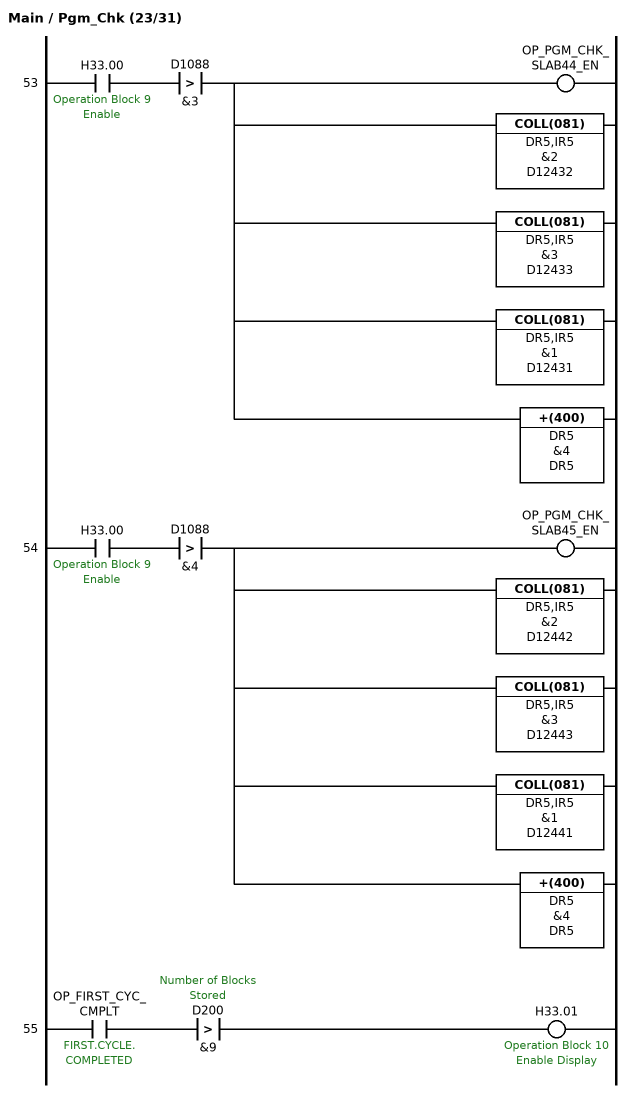
; [picture p120: Main / Pgm_Chk, rungs 53-55]
; rung 53
LD H33.00  ; Operation Block 9 Enable
AND>(320) D1088 &3
OUT OP_PGM_CHK_SLAB44_EN
COLL(081) DR5,IR5 &2 D12432
COLL(081) DR5,IR5 &3 D12433
COLL(081) DR5,IR5 &1 D12431
+(400) DR5 &4 DR5
; rung 54
LD H33.00  ; Operation Block 9 Enable
AND>(320) D1088 &4
OUT OP_PGM_CHK_SLAB45_EN
COLL(081) DR5,IR5 &2 D12442
COLL(081) DR5,IR5 &3 D12443
COLL(081) DR5,IR5 &1 D12441
+(400) DR5 &4 DR5
; rung 55
LD OP_FIRST_CYC_CMPLT  ; FIRST.CYCLE.COMPLETED
AND>(320) D200 &9  ; Number of Blocks Stored
OUT H33.01  ; Operation Block 10 Enable Display

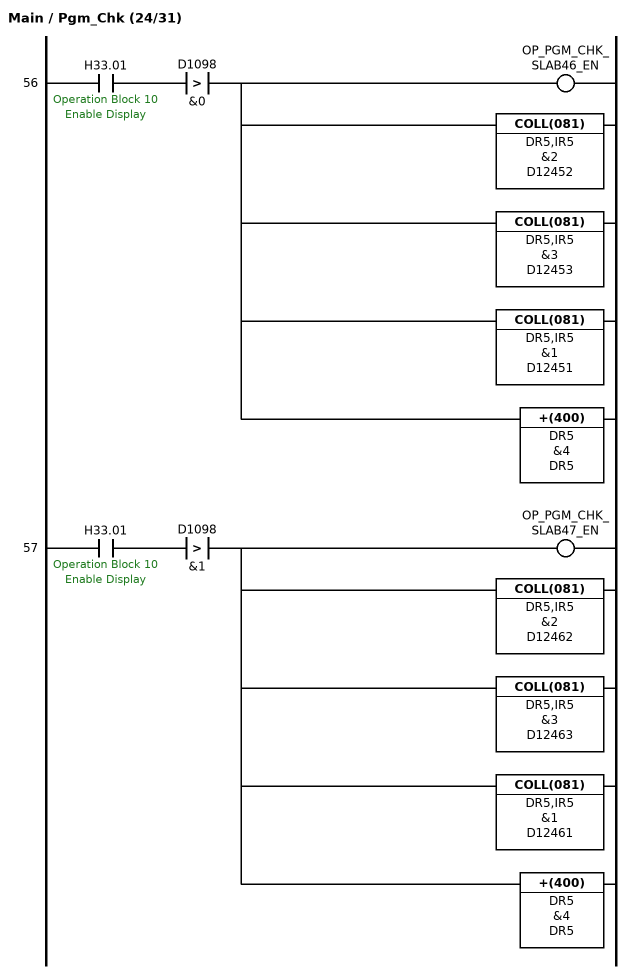
; rung 56
LD H33.01  ; Operation Block 10 Enable Display
AND>(320) D1098 &0
OUT OP_PGM_CHK_SLAB46_EN
COLL(081) DR5,IR5 &2 D12452
COLL(081) DR5,IR5 &3 D12453
COLL(081) DR5,IR5 &1 D12451
+(400) DR5 &4 DR5
; rung 57
LD H33.01  ; Operation Block 10 Enable Display
AND>(320) D1098 &1
OUT OP_PGM_CHK_SLAB47_EN
COLL(081) DR5,IR5 &2 D12462
COLL(081) DR5,IR5 &3 D12463
COLL(081) DR5,IR5 &1 D12461
+(400) DR5 &4 DR5

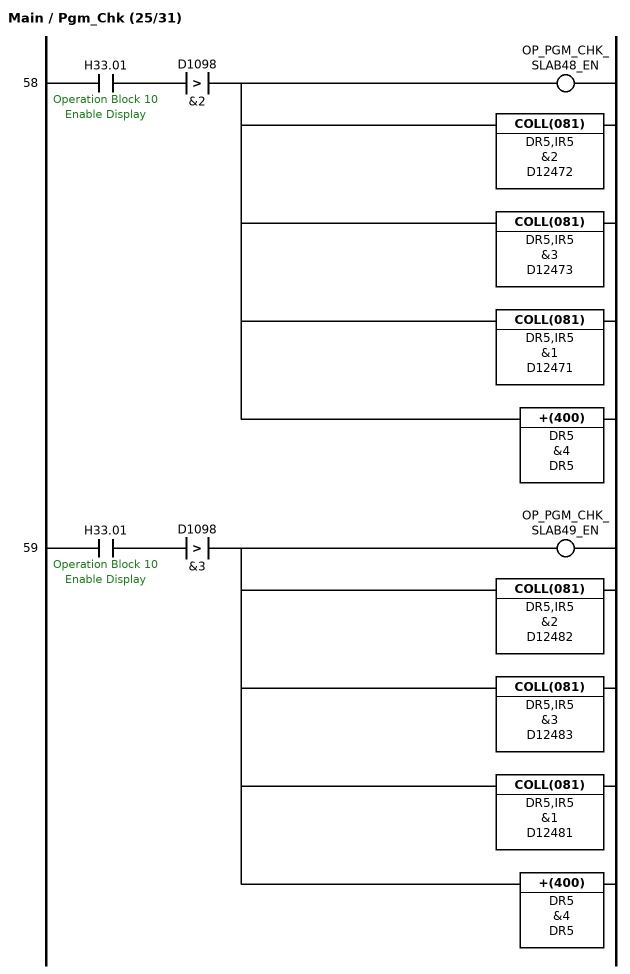
; rung 58
LD H33.01  ; Operation Block 10 Enable Display
AND>(320) D1098 &2
OUT OP_PGM_CHK_SLAB48_EN
COLL(081) DR5,IR5 &2 D12472
COLL(081) DR5,IR5 &3 D12473
COLL(081) DR5,IR5 &1 D12471
+(400) DR5 &4 DR5
; rung 59
LD H33.01  ; Operation Block 10 Enable Display
AND>(320) D1098 &3
OUT OP_PGM_CHK_SLAB49_EN
COLL(081) DR5,IR5 &2 D12482
COLL(081) DR5,IR5 &3 D12483
COLL(081) DR5,IR5 &1 D12481
+(400) DR5 &4 DR5

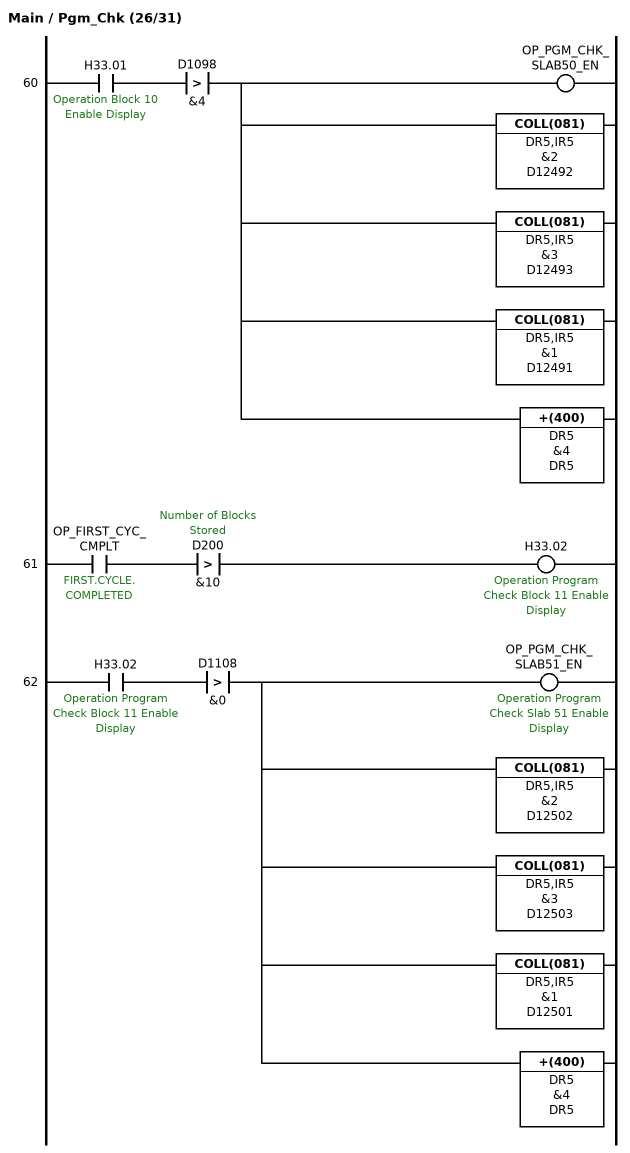
; rung 60
LD H33.01  ; Operation Block 10 Enable Display
AND>(320) D1098 &4
OUT OP_PGM_CHK_SLAB50_EN
COLL(081) DR5,IR5 &2 D12492
COLL(081) DR5,IR5 &3 D12493
COLL(081) DR5,IR5 &1 D12491
+(400) DR5 &4 DR5
; rung 61
LD OP_FIRST_CYC_CMPLT  ; FIRST.CYCLE.COMPLETED
AND>(320) D200 &10  ; Number of Blocks Stored
OUT H33.02  ; Operation Program Check Block 11 Enable Display
; rung 62
LD H33.02  ; Operation Program Check Block 11 Enable Display
AND>(320) D1108 &0
OUT OP_PGM_CHK_SLAB51_EN  ; Operation Program Check Slab 51 Enable Display
COLL(081) DR5,IR5 &2 D12502
COLL(081) DR5,IR5 &3 D12503
COLL(081) DR5,IR5 &1 D12501
+(400) DR5 &4 DR5

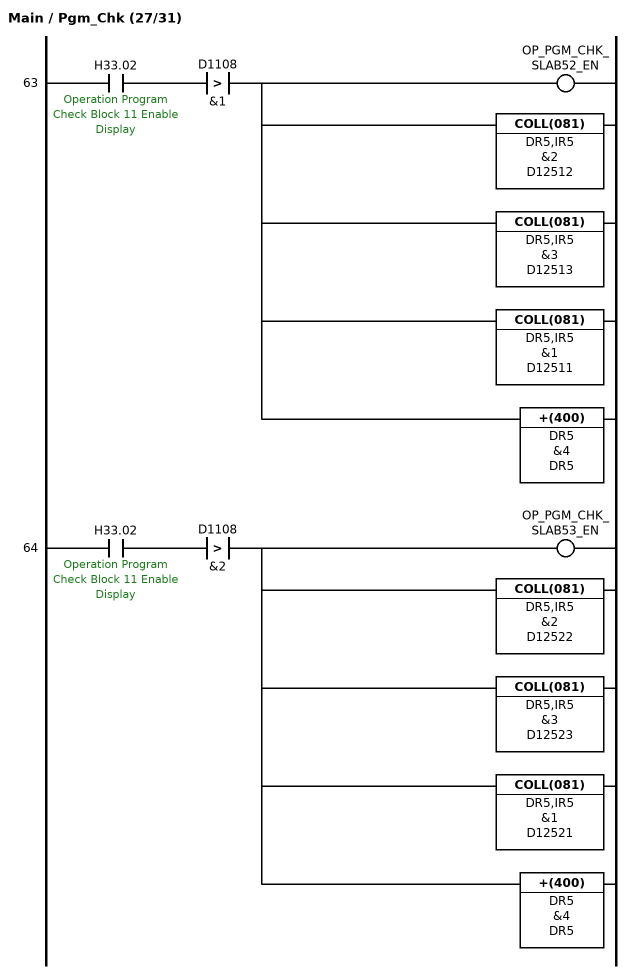
; rung 63
LD H33.02  ; Operation Program Check Block 11 Enable Display
AND>(320) D1108 &1
OUT OP_PGM_CHK_SLAB52_EN
COLL(081) DR5,IR5 &2 D12512
COLL(081) DR5,IR5 &3 D12513
COLL(081) DR5,IR5 &1 D12511
+(400) DR5 &4 DR5
; rung 64
LD H33.02  ; Operation Program Check Block 11 Enable Display
AND>(320) D1108 &2
OUT OP_PGM_CHK_SLAB53_EN
COLL(081) DR5,IR5 &2 D12522
COLL(081) DR5,IR5 &3 D12523
COLL(081) DR5,IR5 &1 D12521
+(400) DR5 &4 DR5

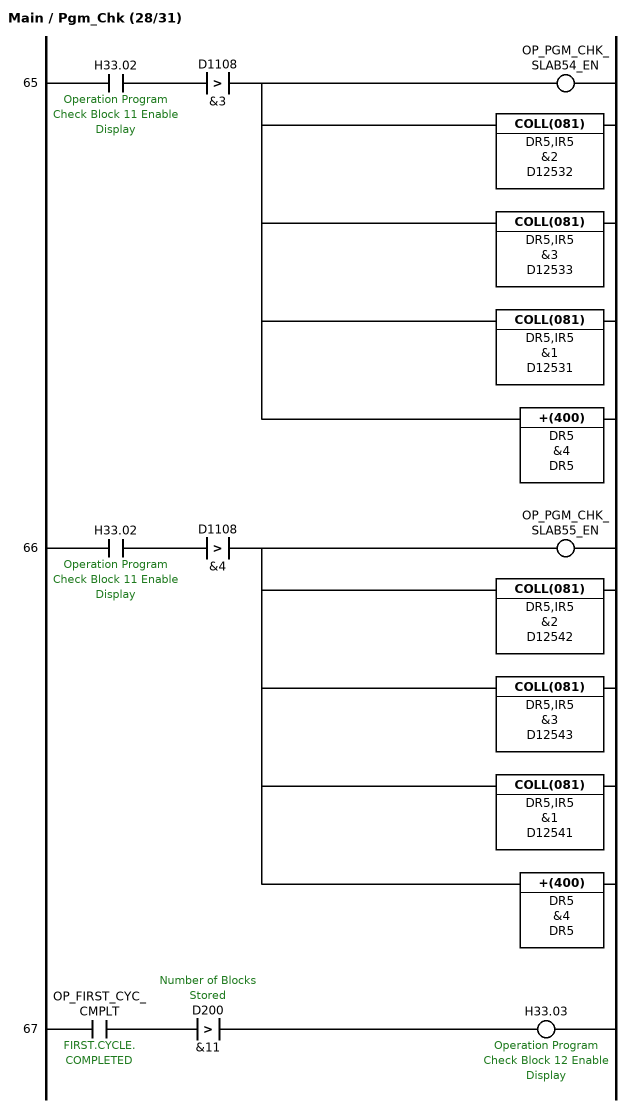
; rung 65
LD H33.02  ; Operation Program Check Block 11 Enable Display
AND>(320) D1108 &3
OUT OP_PGM_CHK_SLAB54_EN
COLL(081) DR5,IR5 &2 D12532
COLL(081) DR5,IR5 &3 D12533
COLL(081) DR5,IR5 &1 D12531
+(400) DR5 &4 DR5
; rung 66
LD H33.02  ; Operation Program Check Block 11 Enable Display
AND>(320) D1108 &4
OUT OP_PGM_CHK_SLAB55_EN
COLL(081) DR5,IR5 &2 D12542
COLL(081) DR5,IR5 &3 D12543
COLL(081) DR5,IR5 &1 D12541
+(400) DR5 &4 DR5
; rung 67
LD OP_FIRST_CYC_CMPLT  ; FIRST.CYCLE.COMPLETED
AND>(320) D200 &11  ; Number of Blocks Stored
OUT H33.03  ; Operation Program Check Block 12 Enable Display

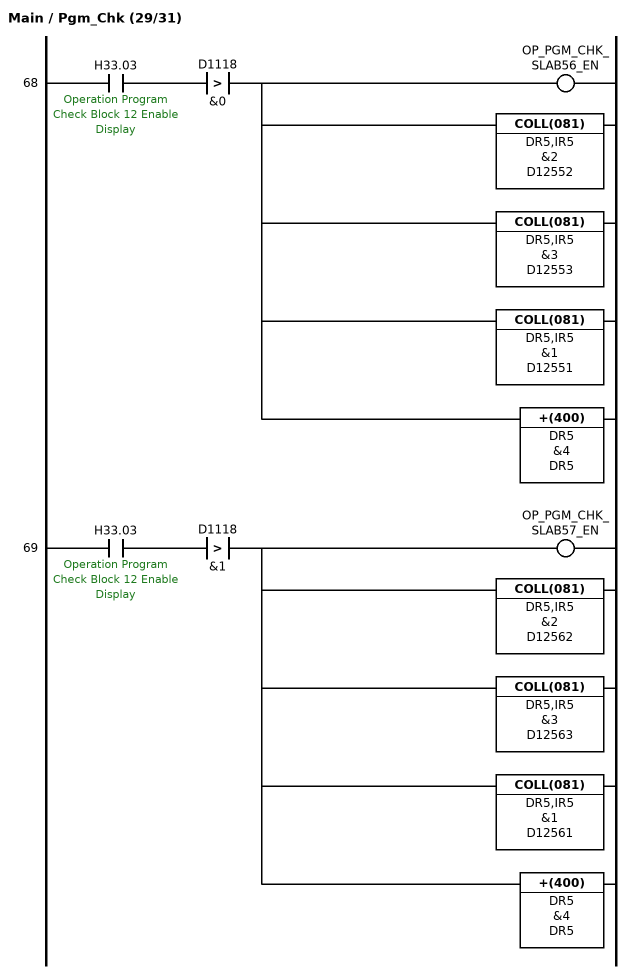
; rung 68
LD H33.03  ; Operation Program Check Block 12 Enable Display
AND>(320) D1118 &0
OUT OP_PGM_CHK_SLAB56_EN
COLL(081) DR5,IR5 &2 D12552
COLL(081) DR5,IR5 &3 D12553
COLL(081) DR5,IR5 &1 D12551
+(400) DR5 &4 DR5
; rung 69
LD H33.03  ; Operation Program Check Block 12 Enable Display
AND>(320) D1118 &1
OUT OP_PGM_CHK_SLAB57_EN
COLL(081) DR5,IR5 &2 D12562
COLL(081) DR5,IR5 &3 D12563
COLL(081) DR5,IR5 &1 D12561
+(400) DR5 &4 DR5

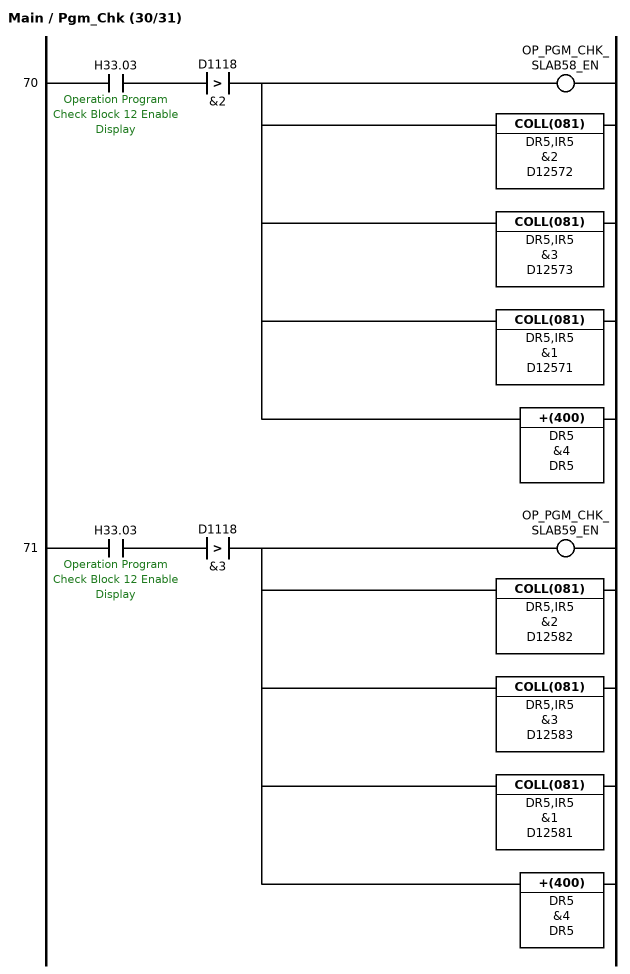
; rung 70
LD H33.03  ; Operation Program Check Block 12 Enable Display
AND>(320) D1118 &2
OUT OP_PGM_CHK_SLAB58_EN
COLL(081) DR5,IR5 &2 D12572
COLL(081) DR5,IR5 &3 D12573
COLL(081) DR5,IR5 &1 D12571
+(400) DR5 &4 DR5
; rung 71
LD H33.03  ; Operation Program Check Block 12 Enable Display
AND>(320) D1118 &3
OUT OP_PGM_CHK_SLAB59_EN
COLL(081) DR5,IR5 &2 D12582
COLL(081) DR5,IR5 &3 D12583
COLL(081) DR5,IR5 &1 D12581
+(400) DR5 &4 DR5

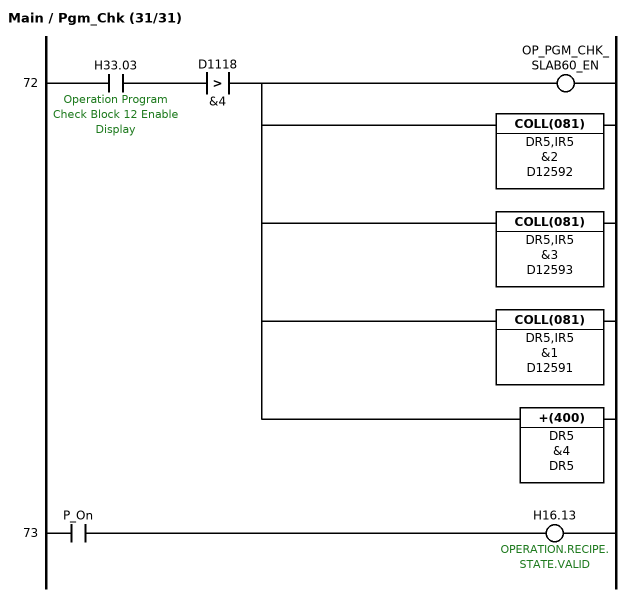
; rung 72
LD H33.03  ; Operation Program Check Block 12 Enable Display
AND>(320) D1118 &4
OUT OP_PGM_CHK_SLAB60_EN
COLL(081) DR5,IR5 &2 D12592
COLL(081) DR5,IR5 &3 D12593
COLL(081) DR5,IR5 &1 D12591
+(400) DR5 &4 DR5
; rung 73
LD P_On
OUT H16.13  ; OPERATION.RECIPE.STATE.VALID

### Section END

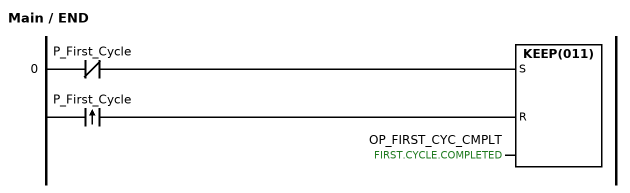
; rung 0
LDNOT P_First_Cycle
@LD P_First_Cycle
KEEP(011) OP_FIRST_CYC_CMPLT  ; FIRST.CYCLE.COMPLETED
; rung 1
END(001)

## Function block Calculate_Pointer
VAR_INPUT
  Word_Count : INT;  (* Number of Words per Record *)
  Offset_Constant : INT;  (* Constant Offset Vaule *)
  Incremet : BOOL;
  Decrement : BOOL;
  Reset_Offset_Pointer : BOOL;  (* Reset Offset and Record Pointers *)
END_VAR
VAR_OUTPUT
  Calculated_Offset : INT;  (* Calculated Offset value *)
  Record_Sel : INT;
  Offset_Calculated : BOOL;  (* Indicates when Offset has been recalculated *)
END_VAR
VAR
  Internal_Count : INT;
  Internal_Calculated_Offset : DINT;
  Internal_Offset_Updated : BOOL;  (* Indicates and update of the offset for use internally. *)
  Internal_Offset_Constant_Compare : INT;  (* Comparison Internal Constant used to trigger a recalulation of the Pointer *)
  Offset_Constant_Changed : BOOL;
  Offset_Calculated_Hold : BOOL;  (* Allow one full scan cycle to complete for the output on time. *)
  TIM100 : BOOL;
END_VAR

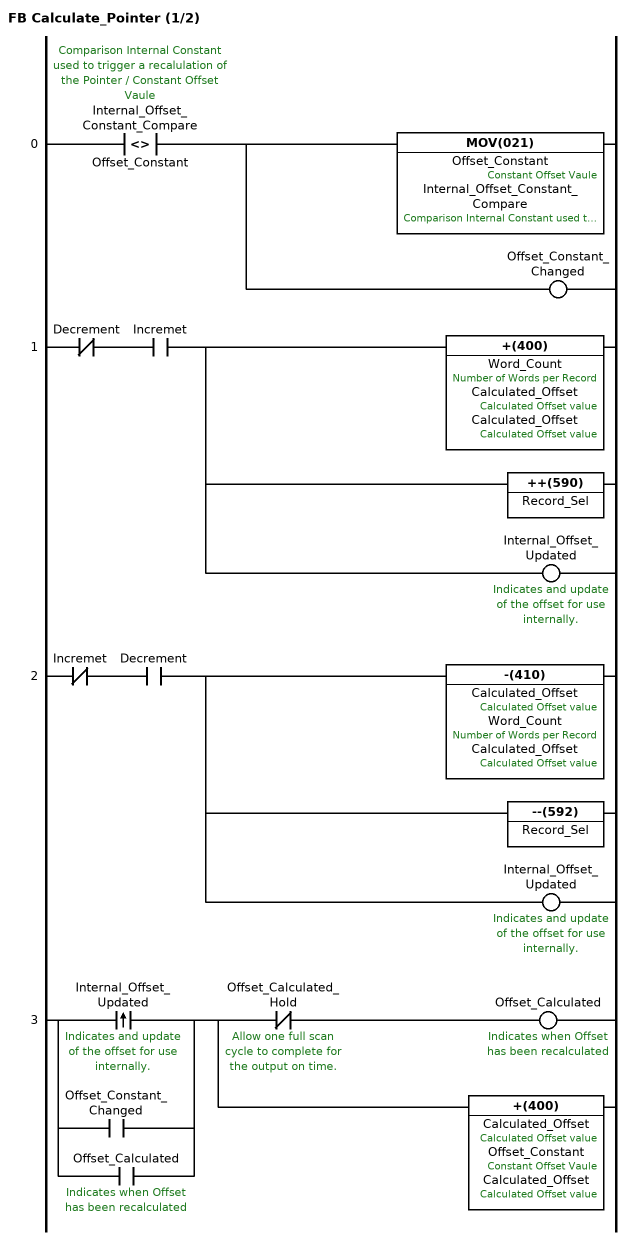
; rung 0
LD<>(305) Internal_Offset_Constant_Compare Offset_Constant  ; Comparison Internal Constant used to trigger a recalulation of the Pointer, Constant Offset Vaule
MOV(021) Offset_Constant Internal_Offset_Constant_Compare  ; Constant Offset Vaule, Comparison Internal Constant used to trigger a recalulation of the Pointer
OUT Offset_Constant_Changed
; rung 1
LDNOT Decrement
AND Incremet
+(400) Word_Count Calculated_Offset Calculated_Offset  ; Number of Words per Record, Calculated Offset value
++(590) Record_Sel
OUT Internal_Offset_Updated  ; Indicates and update of the offset for use internally.
; rung 2
LDNOT Incremet
AND Decrement
-(410) Calculated_Offset Word_Count Calculated_Offset  ; Calculated Offset value, Number of Words per Record
--(592) Record_Sel
OUT Internal_Offset_Updated  ; Indicates and update of the offset for use internally.
; rung 3
@LD Internal_Offset_Updated  ; Indicates and update of the offset for use internally.
OR Offset_Constant_Changed
OR Offset_Calculated  ; Indicates when Offset has been recalculated
OUT TR0
ANDNOT Offset_Calculated_Hold  ; Allow one full scan cycle to complete for the output on time.
OUT Offset_Calculated  ; Indicates when Offset has been recalculated
LD TR0
+(400) Calculated_Offset Offset_Constant Calculated_Offset  ; Calculated Offset value, Constant Offset Vaule

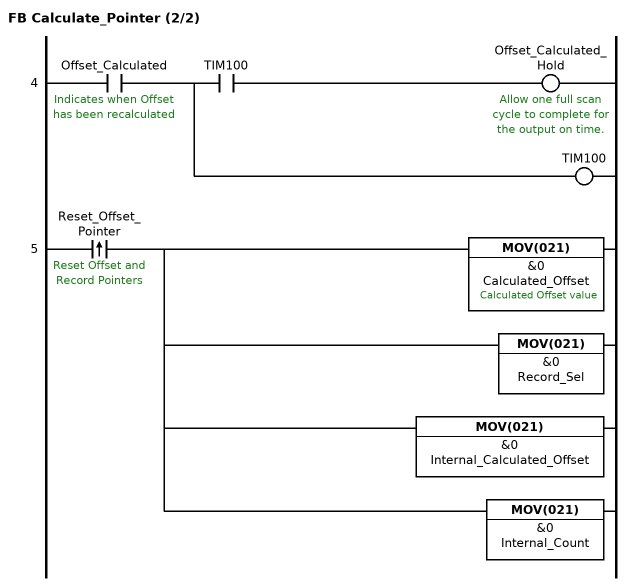
; rung 4
LD Offset_Calculated  ; Indicates when Offset has been recalculated
OUT TR0
AND TIM100
OUT Offset_Calculated_Hold  ; Allow one full scan cycle to complete for the output on time.
LD TR0
OUT TIM100
; rung 5
@LD Reset_Offset_Pointer  ; Reset Offset and Record Pointers
MOV(021) &0 Calculated_Offset  ; Calculated Offset value
MOV(021) &0 Record_Sel
MOV(021) &0 Internal_Calculated_Offset
MOV(021) &0 Internal_Count

## Function block HSC0_INIT
; Initialise HSC Channel Selected
VAR
  Preset : DWORD := 2844843;
END_VAR

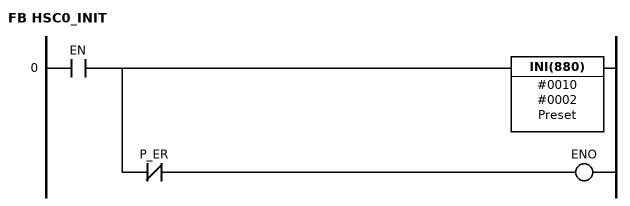
; rung 0
LD EN
INI(880) #0010 #0002 Preset
ANDNOT P_ER
OUT ENO

## Function block HSC1_INIT
; Initialise HSC Channel Selected
VAR
  Preset : DWORD;
END_VAR

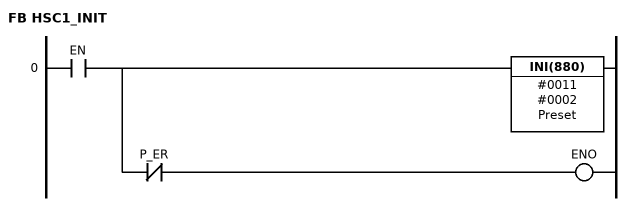
; rung 0
LD EN
INI(880) #0011 #0002 Preset
ANDNOT P_ER
OUT ENO

## Function block MC_Axis_Jog
VAR_INPUT
  jog_plus : BOOL;  (* Jog in the positive direction *)
  jog_minus : BOOL;  (* Jog in the negative direction *)
  ext_err : BOOL;  (* EXTERNAL.ERROR.CONDITION.EXISTS *)
  minus_lim : BOOL;  (* Negative direction limit input *)
  plus_lim : BOOL;  (* Positive direction limit input *)
  JogVelRef : INT;  (* Jog Velocity Reference *)
END_VAR
VAR_OUTPUT
  jog_plus_cmd : BOOL;  (* Jog in the positive direction command *)
  jog_minus_cmd : BOOL;  (* Jog in the negative direction command *)
  jog_active : BOOL;  (* Jog command is active *)
  jog_err : BOOL;  (* Jog error output *)
  JogVelRefCmd : INT;  (* Jog Velocity Reference Command *)
END_VAR
(*Function Block to be used for motion control jogging function*)
ENO:= EN AND NOT ext_err;
jog_err:= ext_err;
JogVelRefCmd:= JogVelRef;
(*Jogging function is available when there is no external error*)
IF NOT ext_err = TRUE THEN 
	(*If either jog button is pressed*)
	IF jog_plus = TRUE OR jog_minus = TRUE THEN jog_active:= TRUE;
		(*If not on plus limit then jog-plus-cmd ok*)
		IF NOT plus_lim = TRUE  THEN jog_plus_cmd:= jog_plus;
		ELSE jog_plus_cmd:= FALSE;
		END_IF;
		IF NOT minus_lim = TRUE THEN jog_minus_cmd:= jog_minus;
		ELSE jog_minus_cmd:= FALSE;
		END_IF;
	ELSE jog_active:= FALSE;
		jog_plus_cmd:= FALSE;
		jog_minus_cmd:= FALSE;
	END_IF;
ELSE jog_active:= FALSE;
	jog_plus_cmd:= FALSE;
	jog_minus_cmd:= FALSE;
END_IF;

## Function block MC_Axis_Motion
VAR_INPUT
  MTN_SAFE : BOOL;  (* Motion is Safe to commence *)
  AXIS_LIM : BOOL;  (* Axis Forard Limit Input *)
  AXIS_MV_TO_POS_CMD : BOOL;  (* Axis Move to Target Position  Command Input *)
  CMD_RST : BOOL;  (* Reset Command *)
  POSN_FDBK : REAL;  (* Axis Position Feedback value in Real format *)
  POSN_CMD : REAL;  (* Axis Position Comanded *)
  POSN_TOL : REAL;  (* Axis in position Tolerance *)
END_VAR
VAR_OUTPUT
  AXIS_MTN_ACT : BOOL;  (* Axis Motion is Active Output *)
  AXIS_MTN_CMD : BOOL;  (* Axis Forward or Index Command (Mode dependant) *)
  AXIS_MTN_CPT : BOOL;  (* Axis Motion Comlete Output *)
  AXIS_IN_POSN : BOOL;  (* Axis in Position Output *)
  AXIS_MTN_ERR : BOOL;  (* Axis Motion Error Output *)
  AXIS_MTN_RDY : BOOL;  (* Axis is Ready for Motion *)
END_VAR
VAR
  POSN_WIN_PLUS : REAL;  (* Axis in Position Window Plus Limit *)
  POSN_WIN_MINUS : REAL;  (* Axis in Position Window Miinus Limit *)
END_VAR
ENO:= EN;
POSN_WIN_PLUS:= POSN_CMD+POSN_TOL;
POSN_WIN_MINUS:= POSN_CMD-POSN_TOL;
IF(MTN_SAFE=TRUE)THEN
	AXIS_MTN_RDY:= TRUE;
ELSE
	AXIS_MTN_RDY:= FALSE;
END_IF;
IF AXIS_MTN_RDY=FALSE AND AXIS_MV_TO_POS_CMD=TRUE THEN
	AXIS_MTN_ERR:= TRUE;
ELSIF AXIS_MTN_RDY = TRUE AND AXIS_MV_TO_POS_CMD = TRUE THEN
	AXIS_MTN_ACT:= TRUE;
	AXIS_MTN_CPT:= FALSE;
END_IF;
IF AXIS_MTN_ACT = TRUE THEN
	IF AXIS_LIM = FALSE AND AXIS_IN_POSN = FALSE THEN
		AXIS_MTN_CMD :=  TRUE;
	ELSE AXIS_MTN_CMD:= FALSE;	
	END_IF;
ELSE AXIS_MTN_CMD:= FALSE;
END_IF;
IF(POSN_FDBK=POSN_CMD) OR (POSN_FDBK <= POSN_WIN_PLUS AND POSN_FDBK >= POSN_WIN_MINUS) AND AXIS_MTN_ACT=TRUE THEN
		AXIS_IN_POSN:= TRUE;
END_IF;
IF(AXIS_IN_POSN=TRUE AND AXIS_MTN_ACT=TRUE)THEN
	AXIS_MTN_CPT:= TRUE;
END_IF;
IF(AXIS_MTN_CPT=TRUE)THEN
	AXIS_MTN_CMD:= FALSE;
	AXIS_MTN_ACT:= FALSE;
END_IF;
IF AXIS_MTN_ERR=TRUE THEN
	AXIS_MTN_ACT:= FALSE;
	AXIS_MTN_CMD:= FALSE;
	AXIS_MTN_CPT:= FALSE;
	AXIS_IN_POSN:= FALSE;
END_IF;
IF(CMD_RST=TRUE)THEN
	AXIS_MTN_CMD:= FALSE;
	AXIS_IN_POSN:= FALSE;
	AXIS_MTN_ERR:= FALSE;
	AXIS_MTN_ACT:= FALSE;
	AXIS_MTN_CPT:= FALSE;
END_IF;

## Function block MC_Axis_Motion_Monitor
VAR_INPUT
  FDBK_POS : REAL;  (* Feedback Position Value in Floating Point *)
  IN_MTN : BOOL;  (* Automatic Mode Selection Enabled *)
  TOLERANCE : REAL;  (* In Position Tolerance *)
END_VAR
VAR_OUTPUT
  FOLLOW_ERR : BOOL;  (* Following Error Condition Exists *)
END_VAR
VAR
  POS_CAPTURED : REAL;  (* Captured Position updated at each scan while motion is happening. If different than feedback, following error output is turned on *)
  TOL_PLUS : REAL;  (* Calculated Plus position based on feedback and tolerance given *)
  TOL_MINUS : REAL;  (* Calculated Minus Position for in position window *)
END_VAR
ENO:= EN;

IF IN_MTN THEN
	
TOL_MINUS:= POS_CAPTURED-TOLERANCE;
TOL_PLUS:= POS_CAPTURED+TOLERANCE;

	IF FDBK_POS > TOL_PLUS OR FDBK_POS < TOL_MINUS THEN
		FOLLOW_ERR:= TRUE;
		POS_CAPTURED:= FDBK_POS;
	ELSE FOLLOW_ERR:= FALSE;
	END_IF;
ELSE
	FOLLOW_ERR:= FALSE;
END_IF;

## Function block MC_Axis_Reset
VAR_INPUT
  RST : BOOL;  (* Axis Reset Command *)
END_VAR
VAR_OUTPUT
  RST_REQ : BOOL;  (* Reset Request *)
END_VAR
(* Reset errored Drive*)
ENO:= EN;
IF(RST) THEN RST_REQ:= TRUE;
ELSE RST_REQ:= FALSE;
END_IF;

## Function block MC_Axis_Srv_Home
VAR_INPUT
  Home_Req : BOOL;  (* Request Homing Sequence *)
  Home_Active : BOOL;  (* Homin command is active *)
  ERR_IN : BOOL;  (* Error monitor *)
  HOME_DN : BOOL;  (* HOME.COMMAND.DONE *)
  INST_TIMER : BOOL;  (* INSTRUCTION EXTERNAL TIMER FOR OVERTIME MONITORING *)
END_VAR
VAR_OUTPUT
  CMD_ACTIVE : BOOL;  (* Command is active *)
  CMD_COMPLETE : BOOL;  (* Command is complete *)
  CMD_ERR : BOOL;  (* Command has errored *)
  HOME_REQ_CMD : BOOL;  (* HOME_REQUEST_COMMAND *)
END_VAR
(*Function Block to be used for motion control Homing function*)
ENO:= EN;
IF (ERR_IN = TRUE) THEN 
	CMD_ERR:= TRUE;
	CMD_ACTIVE:= FALSE;
	CMD_COMPLETE:= FALSE;
	HOME_REQ_CMD:= FALSE;
ELSE
	CMD_ERR:= FALSE;
END_IF;
IF (Home_Req=TRUE ) THEN
	CMD_COMPLETE := FALSE;
	CMD_ACTIVE:= TRUE;
	HOME_REQ_CMD:= TRUE;
ELSIF HOME_DN = TRUE THEN
	CMD_ACTIVE := FALSE;
    HOME_REQ_CMD := FALSE;
    CMD_COMPLETE := TRUE;
END_IF;
IF(INST_TIMER =TRUE) THEN
	CMD_ERR:= TRUE;
	CMD_ACTIVE:= FALSE;
	HOME_REQ_CMD:= FALSE;
	CMD_COMPLETE:= FALSE;
END_IF;

## Function block Op_2_State
VAR_INPUT
  op_state : BOOL;  (* Control Power Status Input from process. *)
END_VAR
VAR_OUTPUT
  op_err : BOOL;  (* Control Power Error Status for User Program use. *)
END_VAR
IF (op_state)THEN 
	ENO := TRUE;
	op_err:= FALSE;
ELSE 
	ENO:=FALSE;
	op_err:= TRUE;
END_IF;

## Function block Op_Alarm_Monitor
VAR_INPUT
  Alm_Monitor_1 : BOOL;  (* Alarm Monitor 1 input *)
  Alm_Monitor_2 : BOOL;  (* Alarm Monitor 2 Input *)
  Alm_Monitor_3 : BOOL;  (* Alarm Monitor 3 Input *)
  Alm_Monitor_4 : BOOL;  (* Alarm Monitor 4 Input *)
  Alm_Monitor_5 : BOOL;  (* Alarm Monitor 5 Input *)
  Alm_Monitor_6 : BOOL;  (* Alarm Monitor 6 Input *)
  Alm_Monitor_7 : BOOL;  (* Alarm Monitor 7 Input *)
  Alm_Monitor_8 : BOOL;  (* Alarm Monitor 8 Input *)
  Alm_Monitor_9 : BOOL;  (* Alarm Monitor 9 Input *)
  Alm_Monitor_10 : BOOL;  (* Alarm Monitor 10 Input *)
  Alm_Monitor_11 : BOOL;  (* Alarm Monitor 11 Input *)
  Alm_Monitor_12 : BOOL;  (* Alarm Monitor 12 Input *)
  Alm_Monitor_13 : BOOL;  (* Alarm Monitor 13 Input *)
  Alm_Monitor_14 : BOOL;  (* Alarm Monitor 14 Input *)
  Alm_Monitor_15 : BOOL;  (* Alarm Monitor 15 Input *)
  Alm_Monitor_16 : BOOL;  (* Alarm Monitor 16 Input *)
END_VAR
VAR_OUTPUT
  Alarm_State : BOOL;
END_VAR
IF NOT (Alm_Monitor_1 = TRUE OR Alm_Monitor_2 = TRUE OR Alm_Monitor_3 = TRUE OR Alm_Monitor_4 = TRUE OR Alm_Monitor_5 = TRUE OR Alm_Monitor_6 = TRUE OR Alm_Monitor_7 = TRUE OR 
	Alm_Monitor_8 =TRUE OR Alm_Monitor_9 = TRUE OR Alm_Monitor_10 = TRUE OR Alm_Monitor_11 = TRUE OR Alm_Monitor_12 = TRUE OR Alm_Monitor_13 = TRUE OR Alm_Monitor_14 = TRUE OR Alm_Monitor_15 = TRUE OR Alm_Monitor_16 = TRUE) THEN
	ENO :=  TRUE;
	Alarm_State := FALSE;
ELSE
	ENO:= FALSE;
	Alarm_State:= TRUE;
END_IF;

## Function block Op_Cyc_Run
VAR_INPUT
  Cyc_Strt : BOOL;  (* CYCLE.START.INPUT *)
  Cyc_Stp : BOOL;  (* CYCLE.STOP.INPUT *)
  MACH_STP : BOOL;  (* MACHINE.STOP.INPUT *)
  ERR_IN : BOOL;  (* SYSTEM.ERROR.INPUT *)
  RST : BOOL;  (* Reset Cycle Run Function *)
END_VAR
VAR_OUTPUT
  IN_CYC : BOOL;  (* IN.CYCLE.RUN *)
  CYC_ERR : BOOL;  (* CYCLE.ERROR *)
  CYC_MACH_STP_CMD : BOOL;  (* CYCLE.MACHINE.STOP.COMMAND *)
  CYC_STP_CMD : BOOL;  (* CYCLE.STOP.COMMAND *)
END_VAR
VAR
  Cycle_Ran : BOOL;
END_VAR
ENO:= EN;
IF Cyc_Strt = TRUE AND Cycle_Ran = FALSE THEN
	CYC_STP_CMD:= FALSE;
	CYC_ERR:= FALSE;
	CYC_MACH_STP_CMD:= FALSE;
	IN_CYC :=  TRUE;	
END_IF;
IF Cyc_Stp = TRUE THEN
	Cycle_Ran:= TRUE;
	IN_CYC:= FALSE;
	CYC_ERR:= FALSE;
	CYC_MACH_STP_CMD:= FALSE;
	CYC_STP_CMD:= TRUE;
END_IF;
IF MACH_STP = TRUE THEN
	Cycle_Ran:= TRUE;
	IN_CYC:= FALSE;
	CYC_STP_CMD:= FALSE;
	CYC_MACH_STP_CMD := TRUE;
ELSE CYC_MACH_STP_CMD :=FALSE;
END_IF;
IF ERR_IN = TRUE THEN
	Cycle_Ran:= FALSE;
	IN_CYC:= FALSE;
	CYC_STP_CMD:= FALSE;
	CYC_ERR:= TRUE;
	CYC_MACH_STP_CMD:= TRUE;
END_IF;
IF RST = TRUE THEN
	Cycle_Ran:= FALSE;
	IN_CYC:= FALSE;
	CYC_STP_CMD:= FALSE;
	CYC_ERR:= FALSE;
	CYC_MACH_STP_CMD:= FALSE;
END_IF;
IF IN_CYC = TRUE AND Cycle_Ran =TRUE THEN 
	IN_CYC:= FALSE;
	Cycle_Ran:= FALSE;
END_IF;

## Function block Op_Cyc_Stp
VAR_INPUT
  Init_Req : BOOL;  (* INITIATE.CYCLE.STOP.REQUEST *)
  In_Cyc_Stp : BOOL;  (* IN.CYCLE.STOP.MONITOR *)
  ERR_IN : BOOL;  (* SYSTEM.ERROR.MONITOR *)
  Res : BOOL;  (* INSTRUCTION.RESET *)
END_VAR
VAR_OUTPUT
  Act : BOOL;  (* CYCLE.STOP.INSTRUCTION.ACTIVE *)
  Cmpt : BOOL;  (* CYCLE.STOP.INSTRUCTION.COMPLETE *)
  Err : BOOL;  (* CYCLE.STOP.INSTRUCTION.ERROR *)
END_VAR
ENO:= EN;
IF Init_Req = TRUE THEN
	Act := TRUE;
	Cmpt:= FALSE;
END_IF;
IF In_Cyc_Stp = TRUE THEN
	Act := FALSE;
	Cmpt := TRUE;
END_IF;
IF ERR_IN = TRUE THEN
	Err := TRUE;
	Act := FALSE;
	Cmpt := FALSE;
END_IF;
IF Res = TRUE THEN 
	Err := FALSE;
	Act := FALSE;
	Cmpt := FALSE;
END_IF;

## Function block Op_Cyc_Strt
VAR_INPUT
  Init_Req : BOOL;  (* INITIATE.START.REQUEST *)
  In_Cyc : BOOL;  (* IN.CYCLE.INPUT *)
  ERR_IN : BOOL;  (* SYSTEM.ERROR.IN.MONITOR *)
  Res : BOOL;  (* RESET.INSTRUCTION *)
END_VAR
VAR_OUTPUT
  Act : BOOL;  (* INSTRUCTION.ACTIVE *)
  Cmpt : BOOL;  (* INSTRUCTION.COMPLETE *)
  Err : BOOL;  (* INSTRUCTION.ERROR *)
END_VAR
ENO := EN;
IF Init_Req = TRUE THEN
	Act := TRUE;
	Cmpt:= FALSE;
END_IF;
IF In_Cyc = TRUE AND Act = TRUE THEN
	Act := FALSE;
	Cmpt := TRUE;
END_IF;
IF ERR_IN = TRUE THEN
	Err := TRUE;
	Act := FALSE;
	Cmpt := FALSE;
END_IF;
IF Cmpt = TRUE AND In_Cyc = FALSE THEN Cmpt:= FALSE;
END_IF;
IF Res = TRUE THEN 
	Err := FALSE;
	Act := FALSE;
	Cmpt := FALSE;
END_IF;

## Function block Op_Cycle_Step
VAR_INPUT
  STATE_VALID : BOOL;  (* Valid State for Stepping Sequence *)
  STATE_INVALID : BOOL;  (* Invalid State for Stepping Sequence *)
  RST : BOOL;  (* Instruction Reset Input *)
END_VAR
VAR_OUTPUT
  STEP_OUT : BOOL;  (* Sequence Step Output Pulse *)
  ERR : BOOL;  (* Error Output *)
END_VAR
ENO:= EN;
IF (STATE_VALID = TRUE AND STATE_INVALID = FALSE) THEN
	STEP_OUT:= TRUE;
	ERR:= FALSE;
ELSIF (STATE_VALID=TRUE AND STATE_INVALID=TRUE) THEN
	STEP_OUT:= FALSE;
	ERR:= TRUE;
ELSIF (STATE_VALID=FALSE AND STATE_INVALID=TRUE)THEN
	STEP_OUT:= FALSE;
	ERR:= FALSE;
END_IF;
IF (RST=TRUE)THEN
	ERR:= FALSE;
END_IF;

## Function block Op_Message
VAR_INPUT
  Message_Select : INT;  (* Select Message to Display *)
  Message_Trigger : BOOL;  (* Trigger Message Change *)
  Message_Colour : INT;  (* Select Message Text Colour *)
END_VAR
VAR_OUTPUT
  Message_Display : INT;  (* Message to display *)
  Message_Colour_Set : INT;  (* Message Colour to Display *)
END_VAR
IF(Message_Trigger)THEN
	Message_Display:= Message_Select;
	Message_Colour_Set:= Message_Colour;
END_IF;

## Function block Op_Mode_Ind
VAR_INPUT
  MODE_0 : BOOL;  (* Mode 0 *)
  MODE_1 : BOOL;  (* Mode 1 *)
  ERR_IN : BOOL;  (* Error In *)
  START_IN : BOOL;
  STOP_IN : BOOL;
  CYCLE_IN : BOOL;  (* In cycle input *)
  HOME_ACT : BOOL;  (* Homing is active input *)
END_VAR
VAR_OUTPUT
  IND_0 : BOOL;
  IND_1 : BOOL;
END_VAR
ENO:= EN;
IF (MODE_0) THEN IND_1:= FALSE; 
	IF (ERR_IN) THEN 
		IND_0:= EN AND P_0_1s;
	ELSIF (HOME_ACT) THEN IND_0:= EN AND P_1s;
	ELSE IND_0:= TRUE;
	END_IF;
ELSIF (MODE_1) THEN IND_0:= FALSE;
	IF (ERR_IN) THEN
		IND_1:= EN AND P_0_1s;
	ELSIF (START_IN AND NOT CYCLE_IN) THEN IND_1:= EN AND P_0_2s;
	ELSIF (STOP_IN AND CYCLE_IN) THEN IND_1:= EN AND P_0_2s;
	ELSIF(CYCLE_IN AND NOT START_IN AND NOT STOP_IN) THEN IND_1:= TRUE;
	ELSE IND_1:= EN AND P_1min;
	END_IF;
END_IF;

## Function block Op_Mode_Sel
VAR_INPUT
  Mode_Sel : BOOL;  (* Input to Select Mode *)
END_VAR
VAR_OUTPUT
  Mode_1 : BOOL;  (* Mode 1 selected *)
  Mode_0 : BOOL;  (* Mode 0 selected *)
END_VAR
IF(Mode_Sel) THEN Mode_1:= TRUE;
	Mode_0:= FALSE;
ELSE Mode_1:= FALSE;
	Mode_0:= TRUE;
END_IF;
ENO:= TRUE;

## Function block Op_Sequence_Step_State_Validate
VAR_INPUT
  TEST1 : BOOL;  (* Test Inut 1 *)
  TEST2 : BOOL;  (* Test Input 2 *)
  TEST3 : BOOL;
  TEST4 : BOOL;
  TEST5 : BOOL;
  TEST6 : BOOL;
  TEST7 : BOOL;
  TEST8 : BOOL;
  TEST9 : BOOL;
  TEST10 : BOOL;
  TEST11 : BOOL;
  TEST12 : BOOL;
  TEST13 : BOOL;
  TEST14 : BOOL;
  TEST15 : BOOL;
  TEST16 : BOOL;
END_VAR
VAR_OUTPUT
  VALID_STATE : BOOL;
  INVALID_STATE : BOOL;
END_VAR
ENO:= EN;
IF  (TEST1<>TRUE OR TEST2<>TRUE OR TEST3<>TRUE OR TEST4<>TRUE OR TEST5<>TRUE OR TEST6<>TRUE OR TEST7<>TRUE OR TEST8<>TRUE OR TEST9<>TRUE OR TEST10<>TRUE OR TEST11<>TRUE OR TEST12<>TRUE OR TEST13<>TRUE OR TEST14<>TRUE OR TEST15<>TRUE OR TEST16<>TRUE) THEN
	VALID_STATE:= FALSE;
	INVALID_STATE:= TRUE;
ELSE
	VALID_STATE:= TRUE;
	INVALID_STATE:= FALSE;
END_IF;